TYPE Acquisition_control :
STRUCT
Trigger_Enable			: BIT;
Trigger					: BIT;
Clear_Exposure_Complete	: BIT;
Reserved3				: BIT;
Reserved4				: BIT;
Reserved5				: BIT;
Reserved6				: BIT;
Set_Offline				: BIT;
END_STRUCT
END_TYPE

(* stored: Version 1.1.0.1, ProductVersion 3.1.4024.11
   DUT Acquisition_control: Id {33628763-e1d1-4034-aea9-ca79eb641d7a} *)
